FUNCTION_BLOCK FB_HeatExchanger1 EXTENDS FB_SystemContinous
VAR_INPUT
END_VAR
VAR_OUTPUT
END_VAR
VAR
END_VAR

END_FUNCTION_BLOCK

(* stored: Version 1.1.0.1, ProductVersion 3.1.4024.10
   POU FB_HeatExchanger1: Id {bca56c6b-1b09-4f57-a186-5b7562770c5b}, SpecialFunc None *)
